PROGRAM F_PRESURIZAR
VAR_INPUT
	Func:E_funcio;
END_VAR
VAR
	///Activa
	xActv: BOOL;
	///Fin Funcion
	xFinFunc: BOOL;
	
	xA_VACIADO: BOOL;
	xA_PRESURIZA: BOOL;
	z_xPresuriza: BOOL;
END_VAR

(*Activa funcio *)
xActv:= func.Actv_Funcio;

(*FIN FUNCION*)
				xFinFunc	:=	xActv AND F_DESPRESURIZA.xDESPRESURIZA;

(*ACTIVA SALIDAS*)
z_xPresuriza:= xActv  ;

END_PROGRAM

(* stored: Version 1.1.0.1, ProductVersion 3.1.4024.10
   POU F_PRESURIZAR: Id {e51a0d5c-960d-4f96-8cce-d1733018d4d5}, SpecialFunc None *)
